(* CODESYS project Prova_TON.project

Project tree, tasks and I/O mapping:
  Device : CODESYS Control Win V3, 3S - Smart Software Solutions GmbH, order no. 305021, version 3.5.10.30
    application Application
      libraries: Standard, * (System)
      task MainTask (cyclic, interval t#20ms, priority 1) calls PLC_PRG
      task VISU_TASK (cyclic, interval 100 ms, priority 31) calls VisuElems.Visu_Prg
      program PLC_PRG [FBD]
      visualisation Visualization
  text list GlobalTextList
*)

// Device/Application/PLC_PRG
PROGRAM PLC_PRG
VAR
	Contact1: BOOL := FALSE;
	Coil1: BOOL := FALSE;
	PT1: TIME := T#8s;
	TON_0: TON;
	Value: TIME;
END_VAR

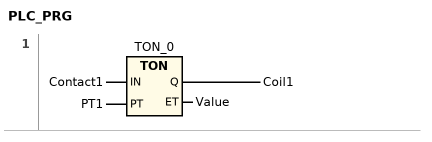
// NETWORK 1
TON_0(IN := Contact1, PT := PT1, ET => Value); // TON
Coil1 := TON_0.Q;

END_PROGRAM

// Device/Application/Visualization
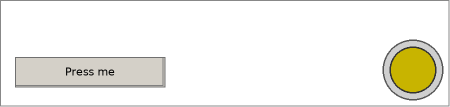
VISUALIZATION Visualization  // 450x107
    Lamp1 (378,35 70x70), variable: PLC_PRG.Coil1, style: Lamp-Lamp1-Yellow
    Button (15,57 150x30), "Press me"
        tap PLC_PRG.Contact1
END_VISUALIZATION
